RoboDK station: Example_01_API - Basics.rdk

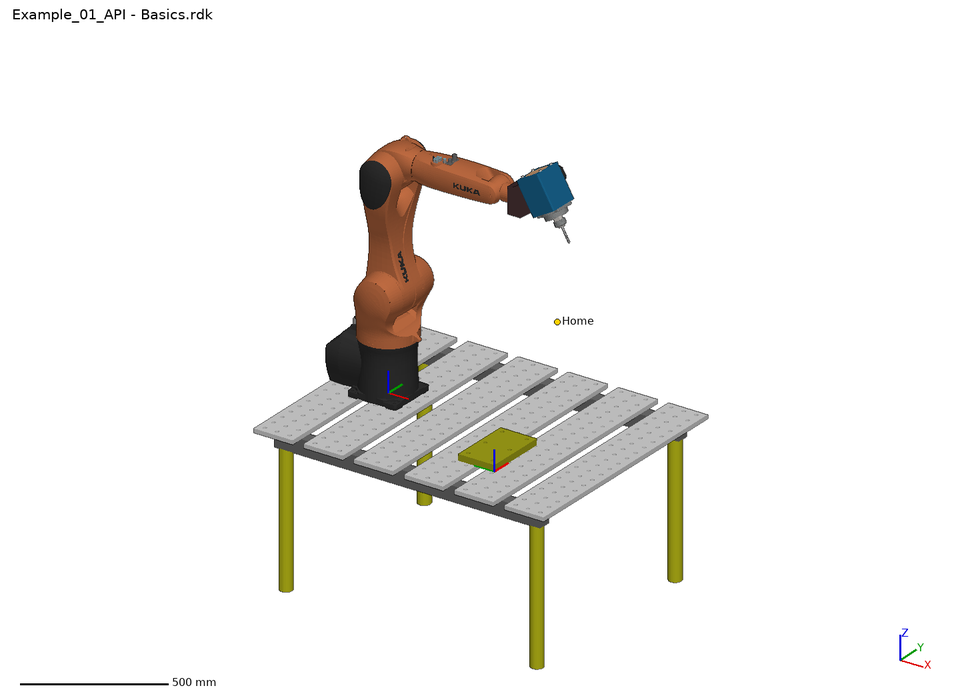
[picture v0: the station drawn from its stored meshes, robots at their saved joint values, targets as dots, program paths as lines]
Station Example_01_API-Basics (saved by RoboDK 5.2.3). Poses are relative to the parent item; angles as X-Y-Z fixed-axis rotations.
  - frame KUKA KR 10 R900 Base at (0, 0, 0) mm
    - robot KUKA KR 10 R900 (model KUKA KR 10 R900 sixx): 6 axes, payload 10 kg, reach 901 mm, repeatability 0.03 mm, weight 52 kg
        modified DH rows (alpha deg, a mm, theta deg, d mm): 0, 0, 0, 400; -90, 25, 0, 0; 0, 455, -90, 0; -90, 35, 0, 420; 90, 0, 0, 0; -90, 0, 180, 80
        joint limits [-170, -190, -120, -185, -120, -350] to [170, 45, 156, 185, 120, 350]; home [0, -90, 90, 0, 0, 0]; saved at [0, -90, 90, 0, 0, 0]
      - tool Spindle, TCP at (116.06, 0, 219.48) mm, rotated rx 0 ry 60 rz 0 deg, size 260.9 x 152 x 222 mm, geometry from Little spindle.step
    - object Table at (380, 0, 0) mm, size 1193.8 x 965.2 x 609.6 mm, geometry from welding_table.sld
  - frame Work Piece at (640.29, -290, 0) mm, rotated rx 0 ry 0 rz 90 deg
    - object Drilling at (0, 0, 0) mm, size 250 x 150 x 25 mm, geometry from Drilling.step
    - target Home (Cartesian target) at (290, -55.8, 461.77) mm, rotated rx -180 ry 0 rz 90 deg; joints [0, -80.983, 104.768, 0, 6.215, 0] of KUKA KR 10 R900
  - Python program Script1 (listed below)

--- Python program Script1 ---
# API to communicate with RoboDK for simulation and offline/online programming
from robodk import *

# Robotics toolbox for industrial robots
from robolink import *

# Start the RoboDK API
# Any connection to RoboDK must be done through Robolink()
# Here we instanciate the Robolink class
RDK = Robolink()

# Force simulation mode in case we are already connected to the robot
RDK.setRunMode(RUNMODE_SIMULATE)

# Retrieving the robot in Station
robot = RDK.Item('',ITEM_TYPE_ROBOT)

REFERENCE_NAME = 'Work Piece'
TARGET_NAME = 'Home'
TOOL_NAME = 'Spindle'

# Get the Reference Frame from station
frame = RDK.Item(REFERENCE_NAME,ITEM_TYPE_FRAME)
if not frame.Valid():
    raise Exception("Reference frame not found. Use name: %s" % REFERENCE_NAME)

# Get the 'Home' target from station
home = RDK.Item(TARGET_NAME, ITEM_TYPE_TARGET)
if not home.Valid():
    raise Exception("Home target is not valid. Set a home target named: %s" % TARGET_NAME)

# Get the tool from station
tool = RDK.Item(TOOL_NAME, ITEM_TYPE_TOOL)
if not tool.Valid():
    raise Exception("Tool is not valid. Use a tool named: %s" % TOOL_NAME)

# List all items in Station Tree
list_items = RDK.ItemList()
for item in list_items:
    print(item.Name())

# Retrieve joints angles for 'Home' Position
jnts = home.Joints()

# Set the robot to the home position
robot.setJoints(jnts)

# Set Robot Speed
robot.setSpeed(200)

# Add a new program
program_name = 'New_Program'
program = RDK.AddProgram(program_name, robot)

# Set Frame
program.setPoseFrame(frame)
# Set Tool
program.setPoseTool(tool)

# Get the pose reference from the home target
pose_ref = robot.Pose()

# Now, we create 3 targets in the station
# Convert the 4x4 pose matrix to XYZABC position
# and orientation angles (mm and deg) from 'Home' position
xyzabc_1 = Pose_2_KUKA(pose_ref)

# Calculating Target 1 by changing Z and orientation
x,y,z,a,b,c = xyzabc_1
xyzabc_2 = [x,y,z+50,a,b,c-45]
target_1 = KUKA_2_Pose(xyzabc_2)

# Calculating Target 2 by changing Y coordinate and orientation
x,y,z,a,b,c = xyzabc_2
xyzabc_3 = [x,y+200,z,a,b,c+40]
target_2 = KUKA_2_Pose(xyzabc_3)

# Calculating Target 3 by changing Z coordinate
# and using Target 2's orientation
xyzabc_4 = Pose_2_KUKA(target_2)
x,y,z,a,b,c = xyzabc_4
xyz_list = [x,y,z+200]
xyz_pose = Mat(target_2) # Create copy of matrix target_2
xyz_pose.setPos(xyz_list)
target_3 = xyz_pose

# Add Target 1 to the Station
T1 = RDK.AddTarget('Target 1', frame)
T1.setPose(target_1)

# Add Target 2 to the Station
T2 = RDK.AddTarget('Target 2', frame)
T2.setPose(target_2)

# Add Target 2 to the Station
T3 = RDK.AddTarget('Target 3', frame)
T3.setPose(target_3)

# First Move instruction of the program as MoveJ
# to avoid initial Singularities
program.MoveJ(T1)
# Using MoveL to move linearly
program.MoveL(T2)
# Using MoveL to move linearly
program.MoveL(T3)

# Generates a Window on RoboDK
RDK.ShowMessage("Program Created in Station", True)
